// TIA Portal V16 export
// export: Created 2021-11-12T13:31:50.1976625Z, ExportSetting WithDefaults, DisplayName Totally Integrated Automation Portal, DisplayVersion V16 Update 3, DisplayName TIA Portal Version Control Interface, DisplayVersion V16 Update 2, DisplayName TIA Portal Openness, DisplayVersion V16 Update 3, DisplayName SINAMICS Startdrive Advanced, DisplayVersion V16 Update 5, DisplayName SINAMICS Startdrive G130, G150, S120, S150, SINAMICS MV, S210, DisplayVersion V16 Update 5, DisplayName SINAMICS Startdrive G110M, G120, G120C, G120D, G120P, G115D, DisplayVersion V16 Update 5, DisplayName STEP 7 Professional, DisplayVersion V16 Update 3, DisplayName STEP 7 Safety, DisplayVersion V16, DisplayName WinCC UA Professional, DisplayVersion V16 Update 3
FUNCTION_BLOCK "IM_000+UH01-KF10"   // FB900, LAD
TITLE = Inputs reading
{ S7_Optimized_Access := 'TRUE' }
VERSION : 0.1
// MICE Wood interface block
// stored: AutoNumber true, IsIECCheckEnabled false, IsRetainMemResEnabled false, MemoryReserve 100, SetENOAutomatically false, UDAEnableTagReadback false
   VAR
      KF11_Ix0 { S7_SetPoint := 'True'} : "STD_CH_DI";
      KF11_Ix1 { S7_SetPoint := 'True'} : "STD_CH_DI";
      KF11_Ix2 { S7_SetPoint := 'True'} : "STD_CH_DI";
      KF11_Ix3 { S7_SetPoint := 'True'} : "STD_CH_DI";
      KF11_Ix4 { S7_SetPoint := 'True'} : "STD_CH_DI";
      KF11_Ix5 { S7_SetPoint := 'True'} : "STD_CH_DI";
      KF11_Ix6 { S7_SetPoint := 'True'} : "STD_CH_DI";
      KF11_Ix7 { S7_SetPoint := 'True'} : "STD_CH_DI";
      KF12_Ix0 { S7_SetPoint := 'True'} : "STD_CH_DI";
      KF12_Ix1 { S7_SetPoint := 'True'} : "STD_CH_DI";
      KF12_Ix2 { S7_SetPoint := 'True'} : "STD_CH_DI";
      KF12_Ix3 { S7_SetPoint := 'True'} : "STD_CH_DI";
      KF12_Ix4 { S7_SetPoint := 'True'} : "STD_CH_DI";
      KF12_Ix5 { S7_SetPoint := 'True'} : "STD_CH_DI";
      KF12_Ix6 { S7_SetPoint := 'True'} : "STD_CH_DI";
      KF12_Ix7 { S7_SetPoint := 'True'} : "STD_CH_DI";
      KF12_Ix8 { S7_SetPoint := 'True'} : "STD_CH_DI";
      KF12_Ix9 { S7_SetPoint := 'True'} : "STD_CH_DI";
      KF12_Ix10 { S7_SetPoint := 'True'} : "STD_CH_DI";
      KF12_Ix11 { S7_SetPoint := 'True'} : "STD_CH_DI";
      KF12_Ix12 { S7_SetPoint := 'True'} : "STD_CH_DI";
      KF12_Ix13 { S7_SetPoint := 'True'} : "STD_CH_DI";
      KF12_Ix14 { S7_SetPoint := 'True'} : "STD_CH_DI";
      KF12_Ix15 { S7_SetPoint := 'True'} : "STD_CH_DI";
      KF13_Ix0 { S7_SetPoint := 'True'} : "STD_CH_DI";
      KF13_Ix1 { S7_SetPoint := 'True'} : "STD_CH_DI";
      KF13_Ix2 { S7_SetPoint := 'True'} : "STD_CH_DI";
      KF13_Ix3 { S7_SetPoint := 'True'} : "STD_CH_DI";
      KF13_Ix4 { S7_SetPoint := 'True'} : "STD_CH_DI";
      KF13_Ix5 { S7_SetPoint := 'True'} : "STD_CH_DI";
      KF13_Ix6 { S7_SetPoint := 'True'} : "STD_CH_DI";
      KF13_Ix7 { S7_SetPoint := 'True'} : "STD_CH_DI";
      KF61_AI0 { S7_SetPoint := 'True'} : "STD_CH_AI";
      KF61_AI1 { S7_SetPoint := 'True'} : "STD_CH_AI";
   END_VAR
   VAR_TEMP   // added for the SCL form of the ladder/FBD networks
      _w1 : Bool;
      _w2 : Bool;
      _w3 : Bool;
      _w4 : Bool;
      _w5 : Bool;
      _w6 : Bool;
      _w7 : Bool;
      _w8 : Bool;
   END_VAR
BEGIN

REGION Network 1: Module position -KF11
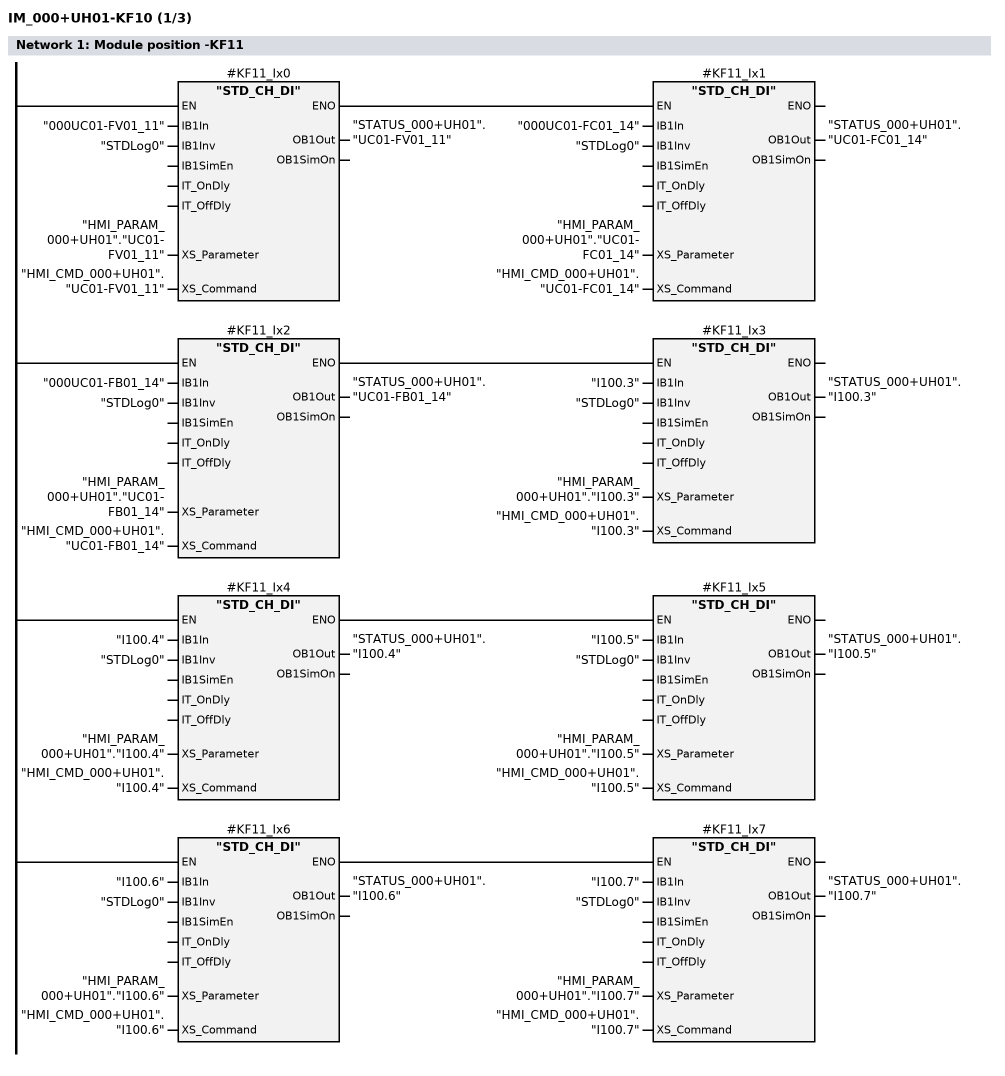
   RUNG wire#powerrail
      #KF11_Ix0(IB1In := "000UC01-FV01_11", IB1Inv := "STDLog0", IB1SimEn :=, IT_OnDly :=, IT_OffDly :=, XS_Parameter := "HMI_PARAM_000+UH01"."UC01-FV01_11", XS_Command := "HMI_CMD_000+UH01"."UC01-FV01_11", OB1Out => "STATUS_000+UH01"."UC01-FV01_11", OB1SimOn =>)
      #KF11_Ix1(IB1In := "000UC01-FC01_14", IB1Inv := "STDLog0", IB1SimEn :=, IT_OnDly :=, IT_OffDly :=, XS_Parameter := "HMI_PARAM_000+UH01"."UC01-FC01_14", XS_Command := "HMI_CMD_000+UH01"."UC01-FC01_14", OB1Out => "STATUS_000+UH01"."UC01-FC01_14", OB1SimOn =>)
   END_RUNG
   RUNG wire#powerrail
      #KF11_Ix2(IB1In := "000UC01-FB01_14", IB1Inv := "STDLog0", IB1SimEn :=, IT_OnDly :=, IT_OffDly :=, XS_Parameter := "HMI_PARAM_000+UH01"."UC01-FB01_14", XS_Command := "HMI_CMD_000+UH01"."UC01-FB01_14", OB1Out => "STATUS_000+UH01"."UC01-FB01_14", OB1SimOn =>)
      #KF11_Ix3(IB1In := "I100.3", IB1Inv := "STDLog0", IB1SimEn :=, IT_OnDly :=, IT_OffDly :=, XS_Parameter := "HMI_PARAM_000+UH01"."I100.3", XS_Command := "HMI_CMD_000+UH01"."I100.3", OB1Out => "STATUS_000+UH01"."I100.3", OB1SimOn =>)
   END_RUNG
   RUNG wire#powerrail
      #KF11_Ix4(IB1In := "I100.4", IB1Inv := "STDLog0", IB1SimEn :=, IT_OnDly :=, IT_OffDly :=, XS_Parameter := "HMI_PARAM_000+UH01"."I100.4", XS_Command := "HMI_CMD_000+UH01"."I100.4", OB1Out => "STATUS_000+UH01"."I100.4", OB1SimOn =>)
      #KF11_Ix5(IB1In := "I100.5", IB1Inv := "STDLog0", IB1SimEn :=, IT_OnDly :=, IT_OffDly :=, XS_Parameter := "HMI_PARAM_000+UH01"."I100.5", XS_Command := "HMI_CMD_000+UH01"."I100.5", OB1Out => "STATUS_000+UH01"."I100.5", OB1SimOn =>)
   END_RUNG
   RUNG wire#powerrail
      #KF11_Ix6(IB1In := "I100.6", IB1Inv := "STDLog0", IB1SimEn :=, IT_OnDly :=, IT_OffDly :=, XS_Parameter := "HMI_PARAM_000+UH01"."I100.6", XS_Command := "HMI_CMD_000+UH01"."I100.6", OB1Out => "STATUS_000+UH01"."I100.6", OB1SimOn =>)
      #KF11_Ix7(IB1In := "I100.7", IB1Inv := "STDLog0", IB1SimEn :=, IT_OnDly :=, IT_OffDly :=, XS_Parameter := "HMI_PARAM_000+UH01"."I100.7", XS_Command := "HMI_CMD_000+UH01"."I100.7", OB1Out => "STATUS_000+UH01"."I100.7", OB1SimOn =>)
   END_RUNG
   // the same network as SCL:
   #KF11_Ix0(IB1In := "000UC01-FV01_11",   // "STD_CH_DI"
             IB1Inv := "STDLog0",
             XS_Parameter := "HMI_PARAM_000+UH01"."UC01-FV01_11",
             XS_Command := "HMI_CMD_000+UH01"."UC01-FV01_11",
             OB1Out => "STATUS_000+UH01"."UC01-FV01_11",
             ENO => #_w1);
   IF #_w1 THEN
       #KF11_Ix1(IB1In := "000UC01-FC01_14",   // "STD_CH_DI"
                 IB1Inv := "STDLog0",
                 XS_Parameter := "HMI_PARAM_000+UH01"."UC01-FC01_14",
                 XS_Command := "HMI_CMD_000+UH01"."UC01-FC01_14",
                 OB1Out => "STATUS_000+UH01"."UC01-FC01_14");
   END_IF;
   #KF11_Ix2(IB1In := "000UC01-FB01_14",   // "STD_CH_DI"
             IB1Inv := "STDLog0",
             XS_Parameter := "HMI_PARAM_000+UH01"."UC01-FB01_14",
             XS_Command := "HMI_CMD_000+UH01"."UC01-FB01_14",
             OB1Out => "STATUS_000+UH01"."UC01-FB01_14",
             ENO => #_w2);
   IF #_w2 THEN
       #KF11_Ix3(IB1In := "I100.3",   // "STD_CH_DI"
                 IB1Inv := "STDLog0",
                 XS_Parameter := "HMI_PARAM_000+UH01"."I100.3",
                 XS_Command := "HMI_CMD_000+UH01"."I100.3",
                 OB1Out => "STATUS_000+UH01"."I100.3");
   END_IF;
   #KF11_Ix4(IB1In := "I100.4",   // "STD_CH_DI"
             IB1Inv := "STDLog0",
             XS_Parameter := "HMI_PARAM_000+UH01"."I100.4",
             XS_Command := "HMI_CMD_000+UH01"."I100.4",
             OB1Out => "STATUS_000+UH01"."I100.4",
             ENO => #_w3);
   IF #_w3 THEN
       #KF11_Ix5(IB1In := "I100.5",   // "STD_CH_DI"
                 IB1Inv := "STDLog0",
                 XS_Parameter := "HMI_PARAM_000+UH01"."I100.5",
                 XS_Command := "HMI_CMD_000+UH01"."I100.5",
                 OB1Out => "STATUS_000+UH01"."I100.5");
   END_IF;
   #KF11_Ix6(IB1In := "I100.6",   // "STD_CH_DI"
             IB1Inv := "STDLog0",
             XS_Parameter := "HMI_PARAM_000+UH01"."I100.6",
             XS_Command := "HMI_CMD_000+UH01"."I100.6",
             OB1Out => "STATUS_000+UH01"."I100.6",
             ENO => #_w4);
   IF #_w4 THEN
       #KF11_Ix7(IB1In := "I100.7",   // "STD_CH_DI"
                 IB1Inv := "STDLog0",
                 XS_Parameter := "HMI_PARAM_000+UH01"."I100.7",
                 XS_Command := "HMI_CMD_000+UH01"."I100.7",
                 OB1Out => "STATUS_000+UH01"."I100.7");
   END_IF;
END_REGION

REGION Network 2: Module position -KF12
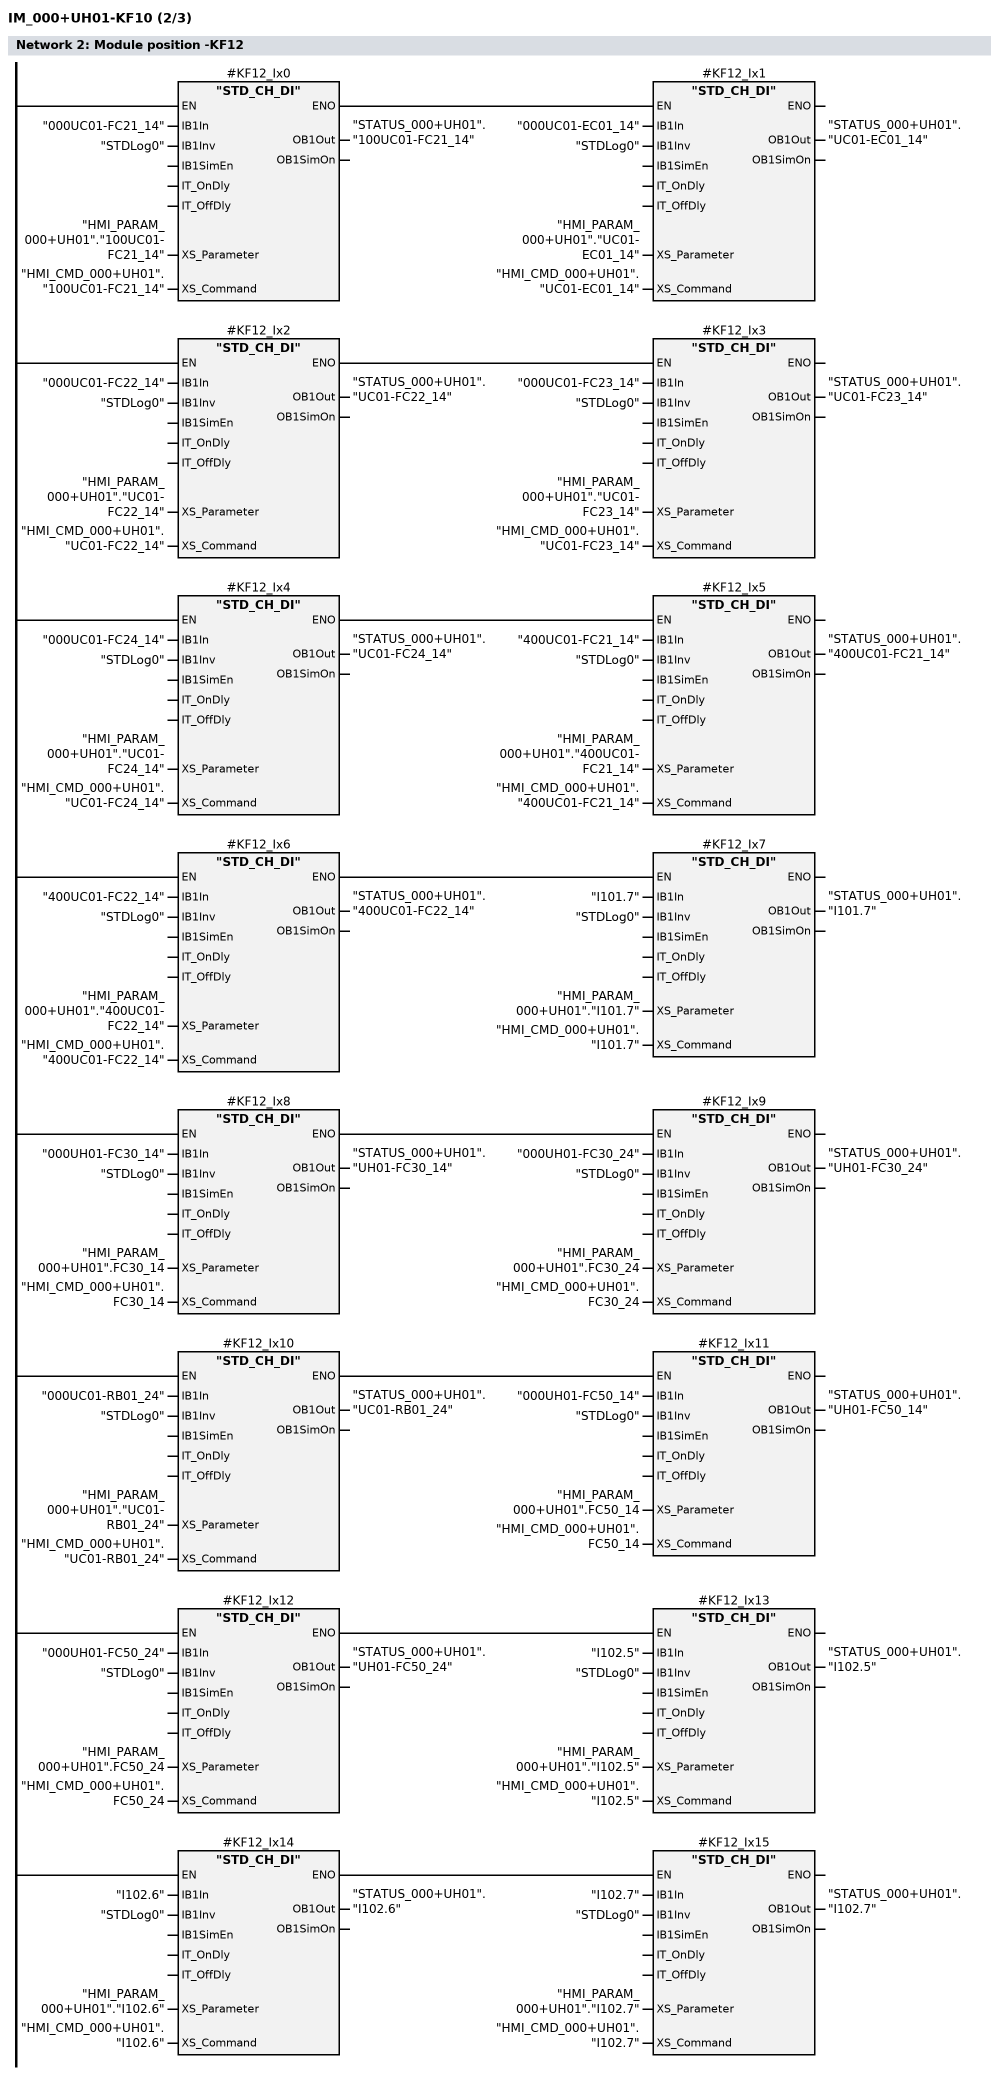
   RUNG wire#powerrail
      #KF12_Ix0(IB1In := "000UC01-FC21_14", IB1Inv := "STDLog0", IB1SimEn :=, IT_OnDly :=, IT_OffDly :=, XS_Parameter := "HMI_PARAM_000+UH01"."100UC01-FC21_14", XS_Command := "HMI_CMD_000+UH01"."100UC01-FC21_14", OB1Out => "STATUS_000+UH01"."100UC01-FC21_14", OB1SimOn =>)
      #KF12_Ix1(IB1In := "000UC01-EC01_14", IB1Inv := "STDLog0", IB1SimEn :=, IT_OnDly :=, IT_OffDly :=, XS_Parameter := "HMI_PARAM_000+UH01"."UC01-EC01_14", XS_Command := "HMI_CMD_000+UH01"."UC01-EC01_14", OB1Out => "STATUS_000+UH01"."UC01-EC01_14", OB1SimOn =>)
   END_RUNG
   RUNG wire#powerrail
      #KF12_Ix2(IB1In := "000UC01-FC22_14", IB1Inv := "STDLog0", IB1SimEn :=, IT_OnDly :=, IT_OffDly :=, XS_Parameter := "HMI_PARAM_000+UH01"."UC01-FC22_14", XS_Command := "HMI_CMD_000+UH01"."UC01-FC22_14", OB1Out => "STATUS_000+UH01"."UC01-FC22_14", OB1SimOn =>)
      #KF12_Ix3(IB1In := "000UC01-FC23_14", IB1Inv := "STDLog0", IB1SimEn :=, IT_OnDly :=, IT_OffDly :=, XS_Parameter := "HMI_PARAM_000+UH01"."UC01-FC23_14", XS_Command := "HMI_CMD_000+UH01"."UC01-FC23_14", OB1Out => "STATUS_000+UH01"."UC01-FC23_14", OB1SimOn =>)
   END_RUNG
   RUNG wire#powerrail
      #KF12_Ix4(IB1In := "000UC01-FC24_14", IB1Inv := "STDLog0", IB1SimEn :=, IT_OnDly :=, IT_OffDly :=, XS_Parameter := "HMI_PARAM_000+UH01"."UC01-FC24_14", XS_Command := "HMI_CMD_000+UH01"."UC01-FC24_14", OB1Out => "STATUS_000+UH01"."UC01-FC24_14", OB1SimOn =>)
      #KF12_Ix5(IB1In := "400UC01-FC21_14", IB1Inv := "STDLog0", IB1SimEn :=, IT_OnDly :=, IT_OffDly :=, XS_Parameter := "HMI_PARAM_000+UH01"."400UC01-FC21_14", XS_Command := "HMI_CMD_000+UH01"."400UC01-FC21_14", OB1Out => "STATUS_000+UH01"."400UC01-FC21_14", OB1SimOn =>)
   END_RUNG
   RUNG wire#powerrail
      #KF12_Ix6(IB1In := "400UC01-FC22_14", IB1Inv := "STDLog0", IB1SimEn :=, IT_OnDly :=, IT_OffDly :=, XS_Parameter := "HMI_PARAM_000+UH01"."400UC01-FC22_14", XS_Command := "HMI_CMD_000+UH01"."400UC01-FC22_14", OB1Out => "STATUS_000+UH01"."400UC01-FC22_14", OB1SimOn =>)
      #KF12_Ix7(IB1In := "I101.7", IB1Inv := "STDLog0", IB1SimEn :=, IT_OnDly :=, IT_OffDly :=, XS_Parameter := "HMI_PARAM_000+UH01"."I101.7", XS_Command := "HMI_CMD_000+UH01"."I101.7", OB1Out => "STATUS_000+UH01"."I101.7", OB1SimOn =>)
   END_RUNG
   RUNG wire#powerrail
      #KF12_Ix8(IB1In := "000UH01-FC30_14", IB1Inv := "STDLog0", IB1SimEn :=, IT_OnDly :=, IT_OffDly :=, XS_Parameter := "HMI_PARAM_000+UH01".FC30_14, XS_Command := "HMI_CMD_000+UH01".FC30_14, OB1Out => "STATUS_000+UH01"."UH01-FC30_14", OB1SimOn =>)
      #KF12_Ix9(IB1In := "000UH01-FC30_24", IB1Inv := "STDLog0", IB1SimEn :=, IT_OnDly :=, IT_OffDly :=, XS_Parameter := "HMI_PARAM_000+UH01".FC30_24, XS_Command := "HMI_CMD_000+UH01".FC30_24, OB1Out => "STATUS_000+UH01"."UH01-FC30_24", OB1SimOn =>)
   END_RUNG
   RUNG wire#powerrail
      #KF12_Ix10(IB1In := "000UC01-RB01_24", IB1Inv := "STDLog0", IB1SimEn :=, IT_OnDly :=, IT_OffDly :=, XS_Parameter := "HMI_PARAM_000+UH01"."UC01-RB01_24", XS_Command := "HMI_CMD_000+UH01"."UC01-RB01_24", OB1Out => "STATUS_000+UH01"."UC01-RB01_24", OB1SimOn =>)
      #KF12_Ix11(IB1In := "000UH01-FC50_14", IB1Inv := "STDLog0", IB1SimEn :=, IT_OnDly :=, IT_OffDly :=, XS_Parameter := "HMI_PARAM_000+UH01".FC50_14, XS_Command := "HMI_CMD_000+UH01".FC50_14, OB1Out => "STATUS_000+UH01"."UH01-FC50_14", OB1SimOn =>)
   END_RUNG
   RUNG wire#powerrail
      #KF12_Ix12(IB1In := "000UH01-FC50_24", IB1Inv := "STDLog0", IB1SimEn :=, IT_OnDly :=, IT_OffDly :=, XS_Parameter := "HMI_PARAM_000+UH01".FC50_24, XS_Command := "HMI_CMD_000+UH01".FC50_24, OB1Out => "STATUS_000+UH01"."UH01-FC50_24", OB1SimOn =>)
      #KF12_Ix13(IB1In := "I102.5", IB1Inv := "STDLog0", IB1SimEn :=, IT_OnDly :=, IT_OffDly :=, XS_Parameter := "HMI_PARAM_000+UH01"."I102.5", XS_Command := "HMI_CMD_000+UH01"."I102.5", OB1Out => "STATUS_000+UH01"."I102.5", OB1SimOn =>)
   END_RUNG
   RUNG wire#powerrail
      #KF12_Ix14(IB1In := "I102.6", IB1Inv := "STDLog0", IB1SimEn :=, IT_OnDly :=, IT_OffDly :=, XS_Parameter := "HMI_PARAM_000+UH01"."I102.6", XS_Command := "HMI_CMD_000+UH01"."I102.6", OB1Out => "STATUS_000+UH01"."I102.6", OB1SimOn =>)
      #KF12_Ix15(IB1In := "I102.7", IB1Inv := "STDLog0", IB1SimEn :=, IT_OnDly :=, IT_OffDly :=, XS_Parameter := "HMI_PARAM_000+UH01"."I102.7", XS_Command := "HMI_CMD_000+UH01"."I102.7", OB1Out => "STATUS_000+UH01"."I102.7", OB1SimOn =>)
   END_RUNG
   // the same network as SCL:
   #KF12_Ix0(IB1In := "000UC01-FC21_14",   // "STD_CH_DI"
             IB1Inv := "STDLog0",
             XS_Parameter := "HMI_PARAM_000+UH01"."100UC01-FC21_14",
             XS_Command := "HMI_CMD_000+UH01"."100UC01-FC21_14",
             OB1Out => "STATUS_000+UH01"."100UC01-FC21_14",
             ENO => #_w1);
   IF #_w1 THEN
       #KF12_Ix1(IB1In := "000UC01-EC01_14",   // "STD_CH_DI"
                 IB1Inv := "STDLog0",
                 XS_Parameter := "HMI_PARAM_000+UH01"."UC01-EC01_14",
                 XS_Command := "HMI_CMD_000+UH01"."UC01-EC01_14",
                 OB1Out => "STATUS_000+UH01"."UC01-EC01_14");
   END_IF;
   #KF12_Ix2(IB1In := "000UC01-FC22_14",   // "STD_CH_DI"
             IB1Inv := "STDLog0",
             XS_Parameter := "HMI_PARAM_000+UH01"."UC01-FC22_14",
             XS_Command := "HMI_CMD_000+UH01"."UC01-FC22_14",
             OB1Out => "STATUS_000+UH01"."UC01-FC22_14",
             ENO => #_w2);
   IF #_w2 THEN
       #KF12_Ix3(IB1In := "000UC01-FC23_14",   // "STD_CH_DI"
                 IB1Inv := "STDLog0",
                 XS_Parameter := "HMI_PARAM_000+UH01"."UC01-FC23_14",
                 XS_Command := "HMI_CMD_000+UH01"."UC01-FC23_14",
                 OB1Out => "STATUS_000+UH01"."UC01-FC23_14");
   END_IF;
   #KF12_Ix4(IB1In := "000UC01-FC24_14",   // "STD_CH_DI"
             IB1Inv := "STDLog0",
             XS_Parameter := "HMI_PARAM_000+UH01"."UC01-FC24_14",
             XS_Command := "HMI_CMD_000+UH01"."UC01-FC24_14",
             OB1Out => "STATUS_000+UH01"."UC01-FC24_14",
             ENO => #_w3);
   IF #_w3 THEN
       #KF12_Ix5(IB1In := "400UC01-FC21_14",   // "STD_CH_DI"
                 IB1Inv := "STDLog0",
                 XS_Parameter := "HMI_PARAM_000+UH01"."400UC01-FC21_14",
                 XS_Command := "HMI_CMD_000+UH01"."400UC01-FC21_14",
                 OB1Out => "STATUS_000+UH01"."400UC01-FC21_14");
   END_IF;
   #KF12_Ix6(IB1In := "400UC01-FC22_14",   // "STD_CH_DI"
             IB1Inv := "STDLog0",
             XS_Parameter := "HMI_PARAM_000+UH01"."400UC01-FC22_14",
             XS_Command := "HMI_CMD_000+UH01"."400UC01-FC22_14",
             OB1Out => "STATUS_000+UH01"."400UC01-FC22_14",
             ENO => #_w4);
   IF #_w4 THEN
       #KF12_Ix7(IB1In := "I101.7",   // "STD_CH_DI"
                 IB1Inv := "STDLog0",
                 XS_Parameter := "HMI_PARAM_000+UH01"."I101.7",
                 XS_Command := "HMI_CMD_000+UH01"."I101.7",
                 OB1Out => "STATUS_000+UH01"."I101.7");
   END_IF;
   #KF12_Ix8(IB1In := "000UH01-FC30_14",   // "STD_CH_DI"
             IB1Inv := "STDLog0",
             XS_Parameter := "HMI_PARAM_000+UH01".FC30_14,
             XS_Command := "HMI_CMD_000+UH01".FC30_14,
             OB1Out => "STATUS_000+UH01"."UH01-FC30_14",
             ENO => #_w5);
   IF #_w5 THEN
       #KF12_Ix9(IB1In := "000UH01-FC30_24",   // "STD_CH_DI"
                 IB1Inv := "STDLog0",
                 XS_Parameter := "HMI_PARAM_000+UH01".FC30_24,
                 XS_Command := "HMI_CMD_000+UH01".FC30_24,
                 OB1Out => "STATUS_000+UH01"."UH01-FC30_24");
   END_IF;
   #KF12_Ix10(IB1In := "000UC01-RB01_24",   // "STD_CH_DI"
              IB1Inv := "STDLog0",
              XS_Parameter := "HMI_PARAM_000+UH01"."UC01-RB01_24",
              XS_Command := "HMI_CMD_000+UH01"."UC01-RB01_24",
              OB1Out => "STATUS_000+UH01"."UC01-RB01_24",
              ENO => #_w6);
   IF #_w6 THEN
       #KF12_Ix11(IB1In := "000UH01-FC50_14",   // "STD_CH_DI"
                  IB1Inv := "STDLog0",
                  XS_Parameter := "HMI_PARAM_000+UH01".FC50_14,
                  XS_Command := "HMI_CMD_000+UH01".FC50_14,
                  OB1Out => "STATUS_000+UH01"."UH01-FC50_14");
   END_IF;
   #KF12_Ix12(IB1In := "000UH01-FC50_24",   // "STD_CH_DI"
              IB1Inv := "STDLog0",
              XS_Parameter := "HMI_PARAM_000+UH01".FC50_24,
              XS_Command := "HMI_CMD_000+UH01".FC50_24,
              OB1Out => "STATUS_000+UH01"."UH01-FC50_24",
              ENO => #_w7);
   IF #_w7 THEN
       #KF12_Ix13(IB1In := "I102.5",   // "STD_CH_DI"
                  IB1Inv := "STDLog0",
                  XS_Parameter := "HMI_PARAM_000+UH01"."I102.5",
                  XS_Command := "HMI_CMD_000+UH01"."I102.5",
                  OB1Out => "STATUS_000+UH01"."I102.5");
   END_IF;
   #KF12_Ix14(IB1In := "I102.6",   // "STD_CH_DI"
              IB1Inv := "STDLog0",
              XS_Parameter := "HMI_PARAM_000+UH01"."I102.6",
              XS_Command := "HMI_CMD_000+UH01"."I102.6",
              OB1Out => "STATUS_000+UH01"."I102.6",
              ENO => #_w8);
   IF #_w8 THEN
       #KF12_Ix15(IB1In := "I102.7",   // "STD_CH_DI"
                  IB1Inv := "STDLog0",
                  XS_Parameter := "HMI_PARAM_000+UH01"."I102.7",
                  XS_Command := "HMI_CMD_000+UH01"."I102.7",
                  OB1Out => "STATUS_000+UH01"."I102.7");
   END_IF;
END_REGION

REGION Network 3: Module position -KF13
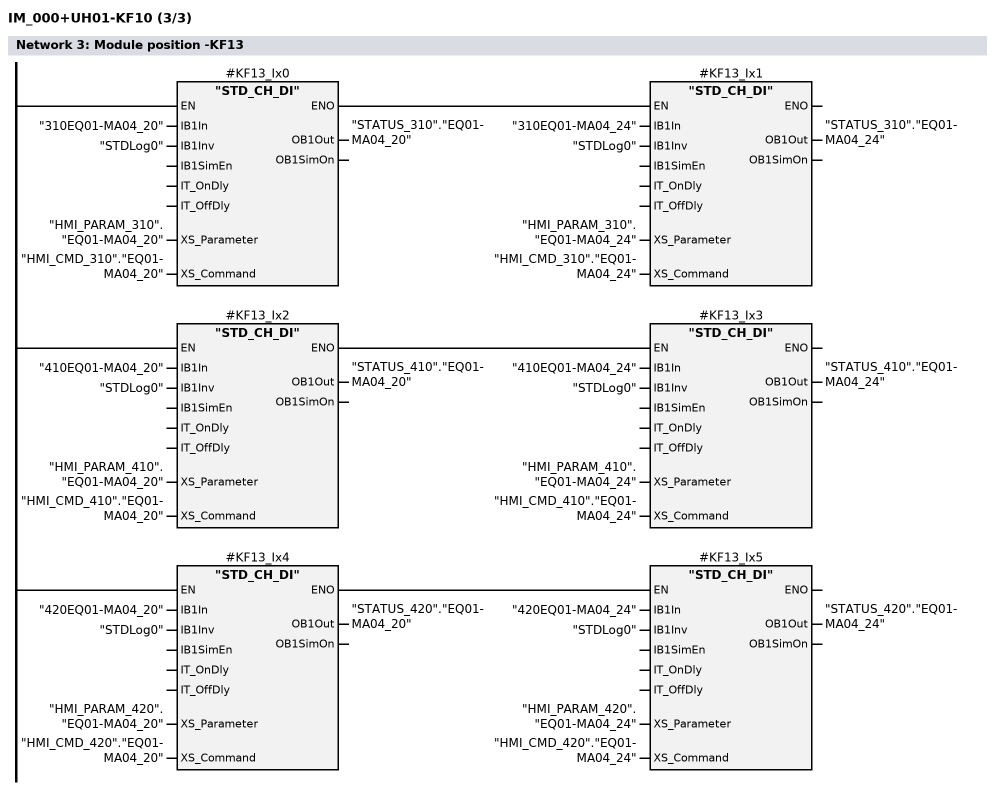
   RUNG wire#powerrail
      #KF13_Ix0(IB1In := "310EQ01-MA04_20", IB1Inv := "STDLog0", IB1SimEn :=, IT_OnDly :=, IT_OffDly :=, XS_Parameter := "HMI_PARAM_310"."EQ01-MA04_20", XS_Command := "HMI_CMD_310"."EQ01-MA04_20", OB1Out => "STATUS_310"."EQ01-MA04_20", OB1SimOn =>)
      #KF13_Ix1(IB1In := "310EQ01-MA04_24", IB1Inv := "STDLog0", IB1SimEn :=, IT_OnDly :=, IT_OffDly :=, XS_Parameter := "HMI_PARAM_310"."EQ01-MA04_24", XS_Command := "HMI_CMD_310"."EQ01-MA04_24", OB1Out => "STATUS_310"."EQ01-MA04_24", OB1SimOn =>)
   END_RUNG
   RUNG wire#powerrail
      #KF13_Ix2(IB1In := "410EQ01-MA04_20", IB1Inv := "STDLog0", IB1SimEn :=, IT_OnDly :=, IT_OffDly :=, XS_Parameter := "HMI_PARAM_410"."EQ01-MA04_20", XS_Command := "HMI_CMD_410"."EQ01-MA04_20", OB1Out => "STATUS_410"."EQ01-MA04_20", OB1SimOn =>)
      #KF13_Ix3(IB1In := "410EQ01-MA04_24", IB1Inv := "STDLog0", IB1SimEn :=, IT_OnDly :=, IT_OffDly :=, XS_Parameter := "HMI_PARAM_410"."EQ01-MA04_24", XS_Command := "HMI_CMD_410"."EQ01-MA04_24", OB1Out => "STATUS_410"."EQ01-MA04_24", OB1SimOn =>)
   END_RUNG
   RUNG wire#powerrail
      #KF13_Ix4(IB1In := "420EQ01-MA04_20", IB1Inv := "STDLog0", IB1SimEn :=, IT_OnDly :=, IT_OffDly :=, XS_Parameter := "HMI_PARAM_420"."EQ01-MA04_20", XS_Command := "HMI_CMD_420"."EQ01-MA04_20", OB1Out => "STATUS_420"."EQ01-MA04_20", OB1SimOn =>)
      #KF13_Ix5(IB1In := "420EQ01-MA04_24", IB1Inv := "STDLog0", IB1SimEn :=, IT_OnDly :=, IT_OffDly :=, XS_Parameter := "HMI_PARAM_420"."EQ01-MA04_24", XS_Command := "HMI_CMD_420"."EQ01-MA04_24", OB1Out => "STATUS_420"."EQ01-MA04_24", OB1SimOn =>)
   END_RUNG
   // the same network as SCL:
   #KF13_Ix0(IB1In := "310EQ01-MA04_20",   // "STD_CH_DI"
             IB1Inv := "STDLog0",
             XS_Parameter := "HMI_PARAM_310"."EQ01-MA04_20",
             XS_Command := "HMI_CMD_310"."EQ01-MA04_20",
             OB1Out => "STATUS_310"."EQ01-MA04_20",
             ENO => #_w1);
   IF #_w1 THEN
       #KF13_Ix1(IB1In := "310EQ01-MA04_24",   // "STD_CH_DI"
                 IB1Inv := "STDLog0",
                 XS_Parameter := "HMI_PARAM_310"."EQ01-MA04_24",
                 XS_Command := "HMI_CMD_310"."EQ01-MA04_24",
                 OB1Out => "STATUS_310"."EQ01-MA04_24");
   END_IF;
   #KF13_Ix2(IB1In := "410EQ01-MA04_20",   // "STD_CH_DI"
             IB1Inv := "STDLog0",
             XS_Parameter := "HMI_PARAM_410"."EQ01-MA04_20",
             XS_Command := "HMI_CMD_410"."EQ01-MA04_20",
             OB1Out => "STATUS_410"."EQ01-MA04_20",
             ENO => #_w2);
   IF #_w2 THEN
       #KF13_Ix3(IB1In := "410EQ01-MA04_24",   // "STD_CH_DI"
                 IB1Inv := "STDLog0",
                 XS_Parameter := "HMI_PARAM_410"."EQ01-MA04_24",
                 XS_Command := "HMI_CMD_410"."EQ01-MA04_24",
                 OB1Out => "STATUS_410"."EQ01-MA04_24");
   END_IF;
   #KF13_Ix4(IB1In := "420EQ01-MA04_20",   // "STD_CH_DI"
             IB1Inv := "STDLog0",
             XS_Parameter := "HMI_PARAM_420"."EQ01-MA04_20",
             XS_Command := "HMI_CMD_420"."EQ01-MA04_20",
             OB1Out => "STATUS_420"."EQ01-MA04_20",
             ENO => #_w3);
   IF #_w3 THEN
       #KF13_Ix5(IB1In := "420EQ01-MA04_24",   // "STD_CH_DI"
                 IB1Inv := "STDLog0",
                 XS_Parameter := "HMI_PARAM_420"."EQ01-MA04_24",
                 XS_Command := "HMI_CMD_420"."EQ01-MA04_24",
                 OB1Out => "STATUS_420"."EQ01-MA04_24");
   END_IF;
END_REGION
END_FUNCTION_BLOCK
